// ---- 7_Visu/Lift_1.TcVIS
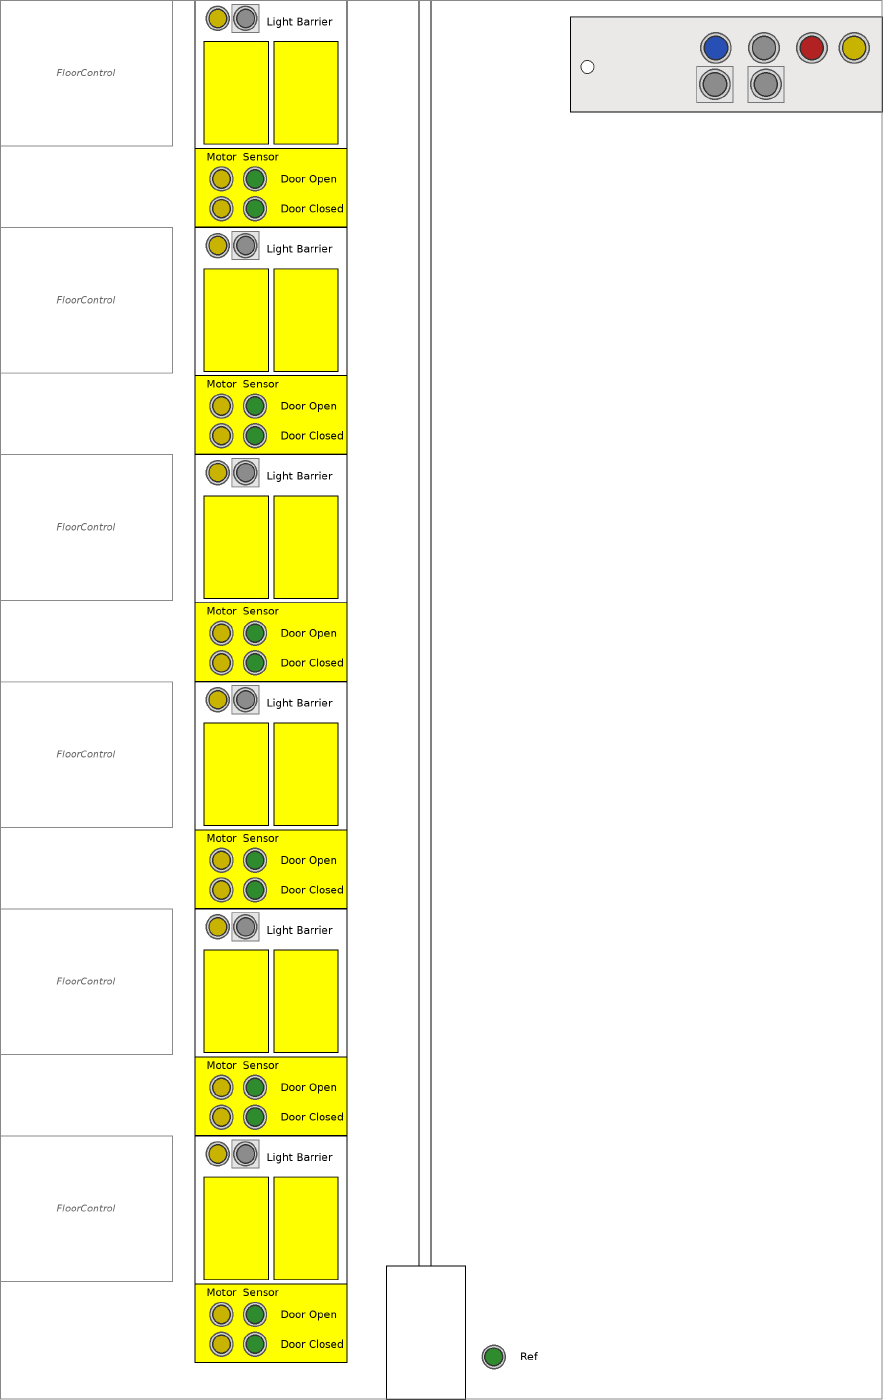
VISUALIZATION Lift_1  // 922x1461
    Frame (0,0 588x1461)
        shows Lift(Position := Visu_L1.Position_LIFT, RefSensor := Visu_L1.Control_LiftAxisReference, Color := Visu_L1.Color, Door_1_Position := Visu_L1.Door_1_Position, Door_1_M_Open := Visu_L1.Door_1_M_Open, Door_1_M_Close := Visu_L1.Door_1_M_Close, Door_2_Position := Visu_L1.Door_2_Position, Door_2_M_Open := Visu_L1.Door_2_M_Open, Door_2_M_Close := Visu_L1.Door_2_M_Close, Door_3_Position := Visu_L1.Door_3_Position, Door_3_M_Open := Visu_L1.Door_3_M_Open, Door_3_M_Close := Visu_L1.Door_3_M_Close, Door_4_Position := Visu_L1.Door_4_Position, Door_4_M_Open := Visu_L1.Door_4_M_Open, Door_4_M_Close := Visu_L1.Door_4_M_Close, Door_5_Position := Visu_L1.Door_5_Position, Door_5_M_Open := Visu_L1.Door_5_M_Open, Door_5_M_Close := Visu_L1.Door_5_M_Close, Door_6_Position := Visu_L1.Door_6_Position, Door_6_M_Open := Visu_L1.Door_6_M_Open, Door_6_M_Close := Visu_L1.Door_6_M_Close, LED_Up_1 := Visu_L1.Panel_1_Led_Up, LED_Down_1 := Visu_L1.Panel_1_Led_Down, FloorNumber_1 := Visu_L1.Panel_1_FloorNumber, BtnLed_1 := Visu_L1.Panel_1_BtnLed, Btn_1 := Visu_L1.Panel_1_Btn, LB_1 := Visu_L1.Door_1_SensorActive, LED_DoorOpen_1 := Visu_L1.Door_1_SensorOpen, LED_DoorClosed_1 := Visu_L1.Door_1_SensorClosed, LED_Up_2 := Visu_L1.Panel_2_Led_Up, LED_Down_2 := Visu_L1.Panel_2_Led_Down, FloorNumber_2 := Visu_L1.Panel_2_FloorNumber, BtnLed_2 := Visu_L1.Panel_2_BtnLed, Btn_2 := Visu_L1.Panel_2_Btn, LB_2 := Visu_L1.Door_2_SensorActive, LED_DoorOpen_2 := Visu_L1.Door_2_SensorOpen, LED_DoorClosed_2 := Visu_L1.Door_2_SensorClosed, LED_Up_3 := Visu_L1.Panel_3_Led_Up, LED_Down_3 := Visu_L1.Panel_3_Led_Down, FloorNumber_3 := Visu_L1.Panel_3_FloorNumber, BtnLed_3 := Visu_L1.Panel_3_BtnLed, Btn_3 := Visu_L1.Panel_3_Btn, LB_3 := Visu_L1.Door_3_SensorActive, LED_DoorOpen_3 := Visu_L1.Door_3_SensorOpen, LED_DoorClosed_3 := Visu_L1.Door_3_SensorClosed, LED_Up_4 := Visu_L1.Panel_4_Led_Up, LED_Down_4 := Visu_L1.Panel_4_Led_Down, FloorNumber_4 := Visu_L1.Panel_4_FloorNumber, BtnLed_4 := Visu_L1.Panel_4_BtnLed, Btn_4 := Visu_L1.Panel_4_Btn, LB_4 := Visu_L1.Door_4_SensorActive, LED_DoorOpen_4 := Visu_L1.Door_4_SensorOpen, LED_DoorClosed_4 := Visu_L1.Door_4_SensorClosed, LED_Up_5 := Visu_L1.Panel_5_Led_Up, LED_Down_5 := Visu_L1.Panel_5_Led_Down, FloorNumber_5 := Visu_L1.Panel_5_FloorNumber, BtnLed_5 := Visu_L1.Panel_5_BtnLed, Btn_5 := Visu_L1.Panel_5_Btn, LB_5 := Visu_L1.Door_5_SensorActive, LED_DoorOpen_5 := Visu_L1.Door_5_SensorOpen, LED_DoorClosed_5 := Visu_L1.Door_5_SensorClosed, LED_Up_6 := Visu_L1.Panel_6_Led_Up, LED_Down_6 := Visu_L1.Panel_6_Led_Down, FloorNumber_6 := Visu_L1.Panel_6_FloorNumber, BtnLed_6 := Visu_L1.Panel_6_BtnLed, Btn_6 := Visu_L1.Panel_6_Btn, LB_6 := Visu_L1.Door_6_SensorActive, LED_DoorOpen_6 := Visu_L1.Door_6_SensorOpen, LED_DoorClosed_6 := Visu_L1.Door_6_SensorClosed)
    Frame (595,17 327x101)
        shows Control(LED_Blue := Visu_L1.Control_LED_Blue, LED_Red := Visu_L1.Control_LED_Red, LED_White := Visu_L1.Control_LED_White, LED_Yellow := Visu_L1.Control_LED_Yellow, Start := Visu_L1.Control_Start, Reset := Visu_L1.Control_Reset, State := Visu_L1.Control_State)
END_VISUALIZATION

// ---- 7_Visu/Handbetrieb.TcVIS
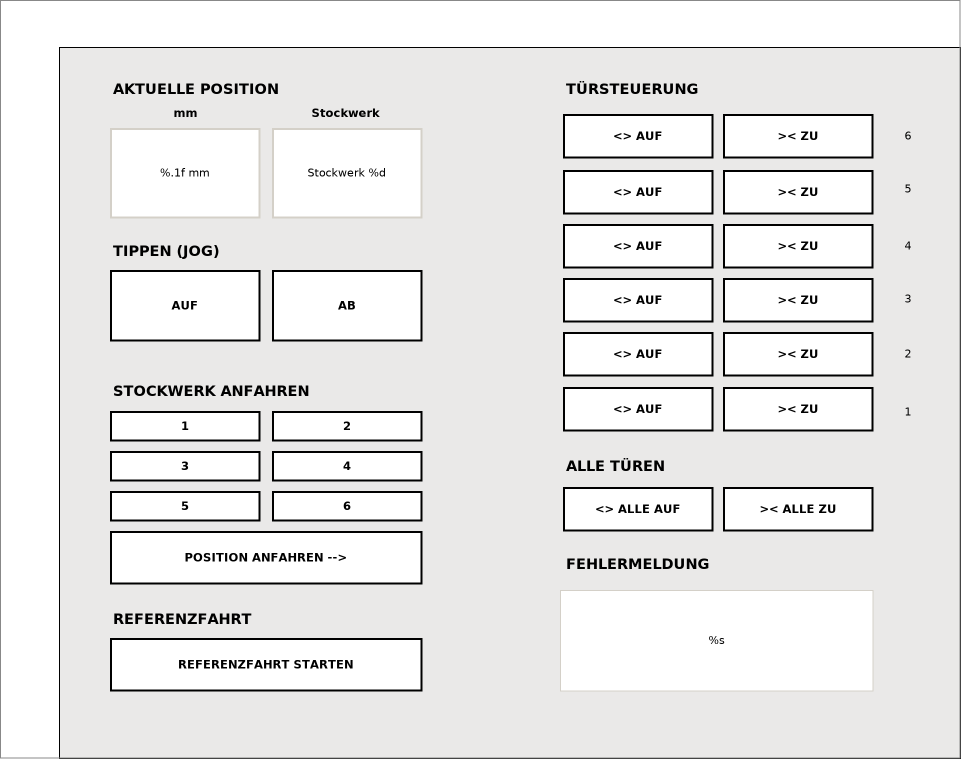
VISUALIZATION Handbetrieb  // 961x759
    RoundedRectangle (59,47 902x712)
    Textfield (110,128 150x90), "%.1f mm", text variable: Divers.AktuellePosmm
    Label (110,74 205x30), "AKTUELLE POSITION"
    Label (110,236 150x30), "TIPPEN (JOG)"
    RoundedRectangle (110,270 150x71), "AUF", colour toggle: Visu_Manuellmodus.JogAuf
        tap Visu_Manuellmodus.JogAuf
    RoundedRectangle (272,270 150x71), "AB", colour toggle: Visu_Manuellmodus.JogAb
        tap Visu_Manuellmodus.JogAb
    Label (110,376 216x30), "STOCKWERK ANFAHREN"
    RoundedRectangle (110,411 150x30), "1", colour variable: Visu_Manuellmodus.adwFloorBtnColor[1]
        OnMouseDown: execute { Visu_Manuellmodus.Zielstock := 1; }
    RoundedRectangle (272,411 150x30), "2", colour variable: Visu_Manuellmodus.adwFloorBtnColor[2]
        OnMouseDown: execute { Visu_Manuellmodus.Zielstock := 2; }
    RoundedRectangle (110,451 150x30), "3", colour variable: Visu_Manuellmodus.adwFloorBtnColor[3]
        OnMouseDown: execute { Visu_Manuellmodus.Zielstock := 3; }
    RoundedRectangle (272,451 150x30), "4", colour variable: Visu_Manuellmodus.adwFloorBtnColor[4]
        OnMouseDown: execute { Visu_Manuellmodus.Zielstock := 4; }
    RoundedRectangle (110,491 150x30), "5", colour variable: Visu_Manuellmodus.adwFloorBtnColor[5]
        OnMouseDown: execute { Visu_Manuellmodus.Zielstock := 5; }
    RoundedRectangle (272,491 150x30), "6", colour variable: Visu_Manuellmodus.adwFloorBtnColor[6]
        OnMouseDown: execute { Visu_Manuellmodus.Zielstock := 6; }
    RoundedRectangle (110,531 312x53), "POSITION ANFAHREN -->"
        tap Visu_Manuellmodus.PosAnfahren
    RoundedRectangle (110,638 312x53), "REFERENZFAHRT STARTEN"
    Label (110,604 150x30), "REFERENZFAHRT"
    Label (563,74 150x30), "TÜRSTEUERUNG"
    RoundedRectangle (563,114 150x44), "<> AUF", colour toggle: Visu_Manuellmodus.bTuerAuf[6]
        tap Visu_Manuellmodus.bTuerAuf[6]
    RoundedRectangle (723,114 150x44), ">< ZU", colour toggle: Visu_Manuellmodus.bTuerZu[6]
        tap Visu_Manuellmodus.bTuerZu[6]
    Label (883,121 50x30), "6"
    Label (883,174 50x30), "5"
    Label (883,231 50x30), "4"
    Label (883,284 50x30), "3"
    Label (883,339 50x30), "2"
    Label (883,397 50x30), "1"
    Label (563,451 150x30), "ALLE TÜREN"
    RoundedRectangle (563,487 150x44), "<> ALLE AUF"
        tap Visu_Manuellmodus.AlleTuerenAuf
    Label (83,98 205x30), "mm"
    Textfield (272,128 150x90), "Stockwerk %d", text variable: Divers.AktuellesStockwerk
    Label (243,98 205x30), "Stockwerk"
    RoundedRectangle (723,487 150x44), ">< ALLE ZU"
        tap Visu_Manuellmodus.AlleTuerenZu
    RoundedRectangle (563,170 150x44), "<> AUF", colour toggle: Visu_Manuellmodus.bTuerAuf[5]
        tap Visu_Manuellmodus.bTuerAuf[5]
    RoundedRectangle (563,224 150x44), "<> AUF", colour toggle: Visu_Manuellmodus.bTuerAuf[4]
        tap Visu_Manuellmodus.bTuerAuf[4]
    RoundedRectangle (563,278 150x44), "<> AUF", colour toggle: Visu_Manuellmodus.bTuerAuf[3]
        tap Visu_Manuellmodus.bTuerAuf[3]
    RoundedRectangle (563,332 150x44), "<> AUF", colour toggle: Visu_Manuellmodus.bTuerAuf[2]
        tap Visu_Manuellmodus.bTuerAuf[2]
    RoundedRectangle (563,387 150x44), "<> AUF", colour toggle: Visu_Manuellmodus.bTuerAuf[1]
        tap Visu_Manuellmodus.bTuerAuf[1]
    RoundedRectangle (723,170 150x44), ">< ZU", colour toggle: Visu_Manuellmodus.bTuerZu[5]
        tap Visu_Manuellmodus.bTuerZu[5]
    RoundedRectangle (723,224 150x44), ">< ZU", colour toggle: Visu_Manuellmodus.bTuerZu[4]
        tap Visu_Manuellmodus.bTuerZu[4]
    RoundedRectangle (723,278 150x44), ">< ZU", colour toggle: Visu_Manuellmodus.bTuerZu[3]
        tap Visu_Manuellmodus.bTuerZu[3]
    RoundedRectangle (723,332 150x44), ">< ZU", colour toggle: Visu_Manuellmodus.bTuerZu[2]
        tap Visu_Manuellmodus.bTuerZu[2]
    RoundedRectangle (723,387 150x44), ">< ZU", colour toggle: Visu_Manuellmodus.bTuerZu[1]
        tap Visu_Manuellmodus.bTuerZu[1]
    Textfield (560,590 313x101), "%s", text variable: Divers.Fehlertext
    Label (563,549 236x30), "FEHLERMELDUNG"
END_VISUALIZATION

// ---- 7_Visu/Visu_Liftkabine.TcVIS
VISUALIZATION Visu_Liftkabine  // 2x2
END_VISUALIZATION

// ---- GlobalTextList.TcGTLO
TEXTLIST GlobalTextList
  252 = '%.1f'
  574 = '%.1f mm'
  227 = '%d'
  25 = '%s'
  836 = '&d'
  819 = '1'
  364 = '2'
  184 = '3'
  881 = '4'
  0 = '5'
  652 = '6'
  839 = '<> ALLE AUF'
  310 = '<> AUF'
  53 = '>< ALLE ZU'
  376 = '>< ZU'
  398 = 'AB'
  383 = 'Aktuelle Position'
  333 = 'AKTUELLE POSITION'
  674 = 'Aktuelle Position in mm'
  220 = 'AKTUELLE POSITION IN MM'
  586 = 'Aktuelles Stockwerk'
  837 = 'ALLE TÜREN'
  769 = 'AUF'
  785 = 'Auf'
  878 = 'Automatic'
  57 = 'Door Closed'
  72 = 'Door Open'
  137 = 'Down'
  349 = 'FEHLERMELDUNG'
  500 = 'Light Barrier'
  230 = 'Ligth Barrier'
  976 = 'Manual'
  812 = 'mm'
  799 = 'Motor'
  204 = 'Off'
  972 = 'POSITION ANFAHREN -->'
  562 = 'Ref'
  253 = 'REFERENZFAHRT'
  434 = 'REFERENZFAHRT DURCHFÜHREN'
  834 = 'REFERENZFAHRT STARTEN'
  488 = 'Sensor'
  735 = 'Stockwerk'
  335 = 'Stockwerk %d'
  820 = 'STOCKWERK ANFAHREN'
  22 = 'TIPPEN (JOG)'
  555 = 'TÜRSTEUERUNG'
  86 = 'Up'
END_TEXTLIST
